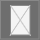
VISUALIZATION VISU_ButtonBack  // 40x40
    RoundedRectangle (0,0 40x40)
        OnMouseClick: change screen: Previous 
    Image (10,5 20x30), image: arrow-return-left_w
        OnMouseClick: change screen: Previous 
END_VISUALIZATION

(* stored: Version 1.1.0.1, ProductVersion 3.1.4024.11
   Visu VISU_ButtonBack: Id {68cd1ca3-c87f-4abe-a6d9-f884257de675} *)
